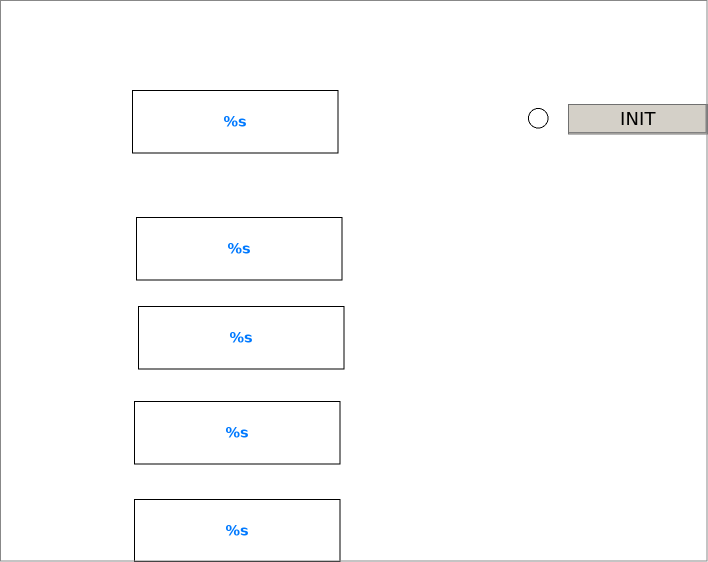
VISUALIZATION Filter_Wheel  // 708x562
    Rectangle (132,90 206x63), "%s", tooltip "Last Command", text variable: MAIN.FILTER_WHEEL.stat.sReply
    Rectangle (136,217 206x63), "%s", tooltip "Last Command", text variable: MAIN.FILTER_WHEEL.stat.sDeviceID
    Rectangle (138,306 206x63), "%s", tooltip "Last Command", text variable: MAIN.FILTER_WHEEL.stat.nCurrentFilterPosition
    Rectangle (134,401 206x63), "%s", tooltip "Last Command", text variable: MAIN.FILTER_WHEEL.stat.sFilterPosition
    Rectangle (134,499 206x63), "%s", tooltip "Last Command", text variable: MAIN.FILTER_WHEEL.stat.bMoveSpeed
    Button (568,104 140x30), "INIT"
        OnMouseClick: execute { MAIN.FILTER_WHEEL.ch_ctrl.nCmd:=E_SA_CH_CMD.REF; }
    Ellipse (528,108 20x20), tooltip "GREEN if initialised", colour toggle: MAIN.FILTER_WHEEL.stat.bInitialised
END_VISUALIZATION

(* stored: Version 1.1.0.1, ProductVersion 3.1.4024.12
   Visu Filter_Wheel: Id {04cdf83d-2d93-4503-8717-ef9187c529cf} *)
